FUNCTION_BLOCK EngToRaw
VAR_INPUT
	iEnabled : BOOL;
	fScaledValue : REAL;
	AnalogConversion : TAnalogConversion;
END_VAR
VAR_OUTPUT
	oEnabled : BOOL;
	wRawValue : WORD;
END_VAR
VAR
END_VAR

//Prepocet z fScaledValue (z PLC) na wRawValue (do procesu po ModbusTCP) podle parametru v AnalogConversion.
wRawValue := REAL_TO_WORD((AnalogConversion.TransducerHiLevel - AnalogConversion.TransducerLoLevel) * (fScaledValue - AnalogConversion.ScaledValLoLevel) / (AnalogConversion.ScaledValHiLevel - AnalogConversion.ScaledValLoLevel) + AnalogConversion.TransducerLoLevel);
oEnabled := iEnabled;

END_FUNCTION_BLOCK

(* stored: Version 1.1.0.1, ProductVersion 3.1.4024.13
   POU EngToRaw: Id {c671cf82-59e0-434c-ac72-b75741f36d84}, SpecialFunc None *)
